{attribute 'qualified_only'}
VAR_GLOBAL
	mb_Input_Coils	:	ARRAY [0..3] OF BOOL;
	mb_Output_Coils	:   ARRAY [0..5] OF BOOL;
END_VAR

(* stored: Version 1.1.0.1, ProductVersion 3.1.4024.12
   GVL GVL: Id {2eeeaaa3-b845-42c5-b044-c9905e71acd7} *)
